PROGRAM P_Demo_LrealIsNaN
VAR
    lrSensor : LREAL;
    bIsNaN   : BOOL;
    bCheck   : BOOL;
END_VAR

// ============================================================
// Tc2_Utilities.LrealIsNaN 演示程序（FUNCTION，单周期触发）
// ============================================================
// 场景：积分器算出 0/0 后变 NaN，在喂下游前判 NaN 切回安全默认值。
// 价值：替代手写 `NOT(x = x)`；语义清晰。
// 验证步骤：
//   1. 把本 PROGRAM 加到 PlcTask 调用列表
//   2. 编译 + 登录
//   3. 在线把 b... 触发位置 TRUE 一个周期
//   4. 观察输出变量是否符合期望
// ============================================================

IF bCheck THEN
    bIsNaN := LrealIsNaN(lrSensor);
    bCheck := FALSE;
END_IF;

END_PROGRAM

(* stored: Version 1.1.0.1, ProductVersion 3.1.4024.5
   POU P_Demo_LrealIsNaN: Id {6ddc7825-0e52-52c0-b897-5c20794c7f4c}, SpecialFunc None *)
